FUNCTION TryConvert_UINT_TO_BYTE : BOOL
VAR_INPUT
	in : UINT;
	out : REFERENCE TO BYTE;
END_VAR

IF in > DatatypeLimits.MAX_VALUE_OF_UINT_WHICH_CAN_BE_HELD_IN_A_BYTE THEN
	RETURN;
END_IF

out := UINT_TO_BYTE(in);
TryConvert_UINT_TO_BYTE := TRUE;

END_FUNCTION

(* stored: Version 1.1.0.1, ProductVersion 3.1.4024.12
   POU TryConvert_UINT_TO_BYTE: Id {d011c2b8-a618-47a9-b190-5c15b0e55dd8}, SpecialFunc None *)
